TYPE CmpWMxFQAGateConfig :
STRUCT
	DBLocation: STRING(30);
END_STRUCT
END_TYPE

(* stored: Version 1.1.0.1, ProductVersion 3.1.4024.6
   DUT CmpWMxFQAGateConfig: Id {c70fa506-0486-413e-971e-e273a50c4c4e} *)
